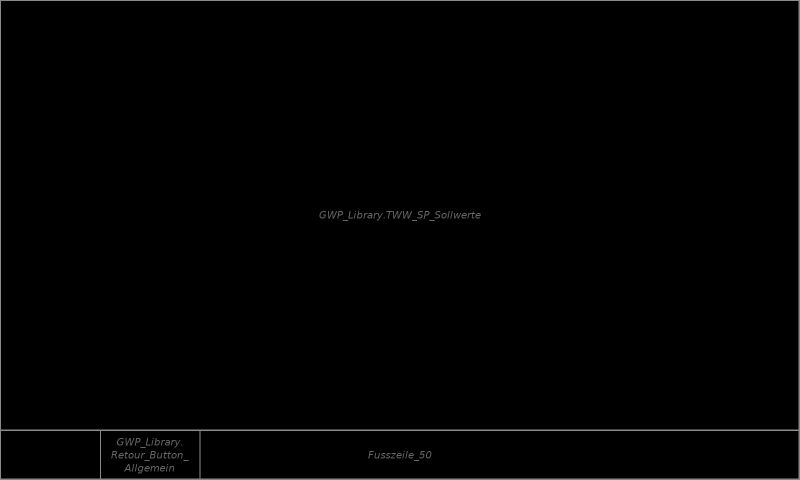
VISUALIZATION TWW_SP_Sollwerte  // 800x480
    Frame (0,0 800x430)
        shows GWP_Library.TWW_SP_Sollwerte(FB_TWW_SP := Main.TWW_SP_0, FB_Kreis_3KO := Main.Kreis_3KO_0)
    Frame (0,430 800x50)
        shows Fusszeile_50()
    Frame (100,430 100x50)
        shows GWP_Library.Retour_Button_Allgemein()
END_VISUALIZATION

(* stored: Version 1.1.0.1, ProductVersion 3.1.4022.6
   Visu TWW_SP_Sollwerte: Id {6321b763-ee9b-4493-ac0b-17b148cd575b} *)
